VAR_GLOBAL CONSTANT
	RS_NUMBER	: UINT := 4;
END_VAR

(* stored: Version 1.1.0.1, ProductVersion 3.1.4024.12
   GVL CONSTANTS: Id {4c0d8cd1-005d-4e3a-9512-f66f848aabc8} *)
